// TIA Portal V16 export
// export: Created 2025-05-30T16:35:54.1073533Z, ExportSetting WithDefaults, DisplayName Totally Integrated Automation Portal, DisplayVersion V16, DisplayName TIA Portal Version Control Interface, DisplayVersion V16, DisplayName TIA Portal Openness, DisplayVersion V16, DisplayName STEP 7 Professional, DisplayVersion V16, DisplayName STEP 7 Safety, DisplayVersion V16, DisplayName WinCC Advanced, DisplayVersion V16
FUNCTION_BLOCK "Ouput_Function_1"   // FB8, FBD
TITLE = Ouput Controller Function Block
VERSION : 0.1
// stored: AutoNumber true, IsIECCheckEnabled false, UDAEnableTagReadback false
   VAR_INPUT
      "Stop Contact" : Bool;
      "Manual Command" : Bool;
      "Auto Command" : Bool;
      "Option Command" : Bool;
      "Disable Command" : Bool;
   END_VAR
   VAR_OUTPUT
      "Ouput Signal" : Bool;
   END_VAR
BEGIN

REGION Network 1: Ouput Controller
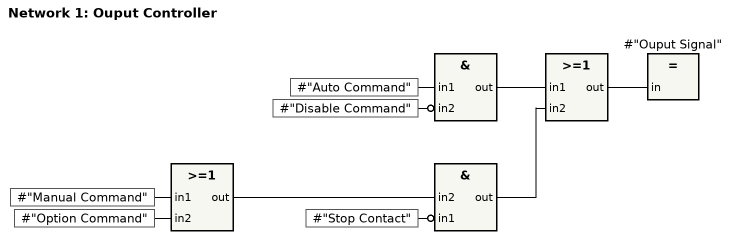
   #"Ouput Signal" := (#"Auto Command" AND NOT #"Disable Command") OR ((#"Manual Command" OR #"Option Command") AND NOT #"Stop Contact");
END_REGION
END_FUNCTION_BLOCK
